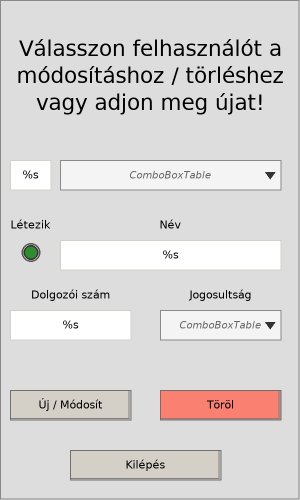
VISUALIZATION AddDelete  // 300x500
    Label (10,10 281x131), "Válasszon felhasználót a módosításhoz / törléshez vagy adjon meg újat!"
    Button (70,450 151x30), "Kilépés"
        toggle GVL.AddDeleteEnabled
    ComboBoxTable (60,160 221x30), variable: GVL.UserID_Temp, data array: GVL.Users
        p3854506369: GVL.Users[INDEX].UserID
        p1892666644: GVL.Users[INDEX].UserNumber
        p338671338: GVL.Users[INDEX].UserName
        p2170511999: GVL.Users[INDEX].UserLevel
        p3723444502: GVL.Users[INDEX].UserExist
    Textfield (10,310 121x30), "%s", text variable: GVL.UserTemp.UserNumber
        OnMouseClick: write the text variable via VisuDialogs.Numpad
    Textfield (60,240 221x30), "%s", text variable: GVL.UserTemp.UserName
        OnMouseClick: write the text variable via Edit
    Button (10,390 121x30), "Új / Módosít"
        toggle GVL.UserModify
    Button (160,390 121x30), "Töröl"
        OnMouseClick: OpenDialog Dialog=Biztos, OpenModal=True, OpenCentered=True
    Label (60,210 221x30), "Név"
    Label (10,280 121x30), "Dolgozói szám"
    Label (160,280 121x30), "Jogosultság"
    Textfield (10,160 41x30), "%s", text variable: GVL.UserTemp.UserID
    Lamp1 (20,240 22x25), variable: GVL.UserTemp.UserExist, style: Lamp-Lamp1-Green
    ComboBoxTable (160,310 121x30), variable: GVL.UserTemp.UserLevel, data array: GVL.UserLevels
        p3854506369: GVL.UserLevels[INDEX]
    Label (10,210 41x30), "Létezik"
END_VISUALIZATION

(* stored: Version 1.1.0.1, ProductVersion 3.1.4024.11
   Visu AddDelete: Id {f205caf7-c621-4fda-a26f-d017ca991b5c} *)
